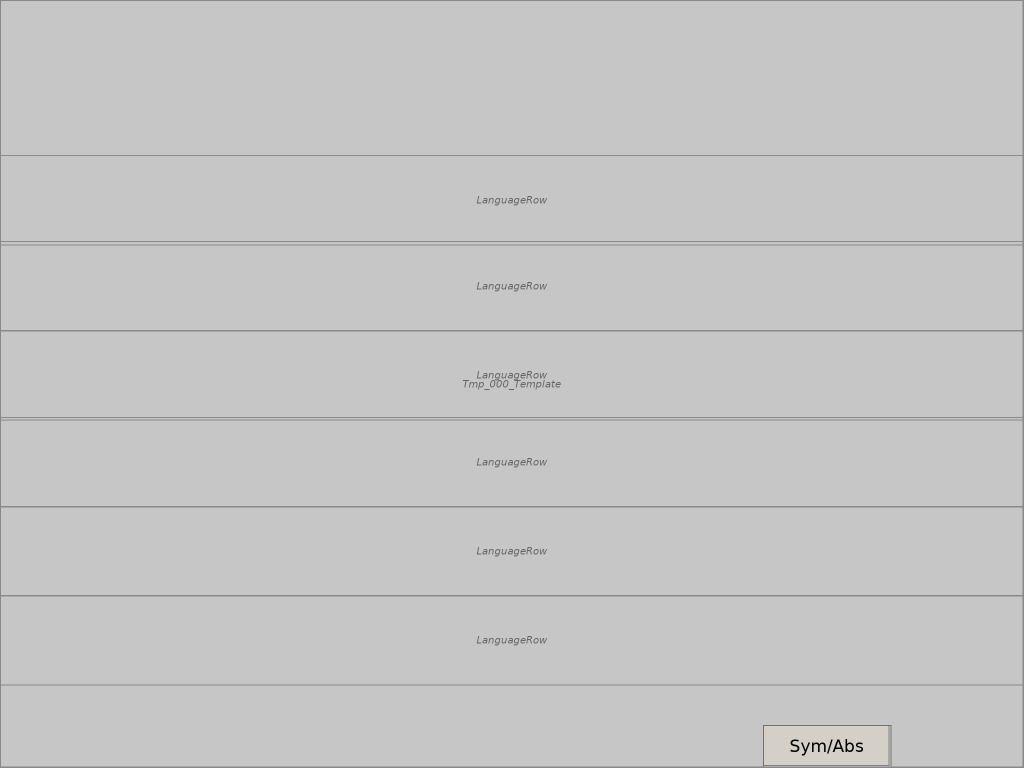
VISUALIZATION Unt_403_Language  // 1024x768
    Frame (0,0 1024x768)
        shows Tmp_000_Template(header := gHMIData.hmiHeader)
    Frame (0,155 1024x90)
        shows LanguageRow(MotionRowInstanceSingle := gHMIData.gLangRows.gMotionRow1, MotionRowButtonsSingle := gHMIData.gLangButtons.gMotionRow1btn)
    Frame (0,241 1024x90)
        shows LanguageRow(MotionRowInstanceSingle := gHMIData.gLangRows.gMotionRow2, MotionRowButtonsSingle := gHMIData.gLangButtons.gMotionRow2btn)
    Frame (0,330 1024x90)
        shows LanguageRow(MotionRowInstanceSingle := gHMIData.gLangRows.gMotionRow3, MotionRowButtonsSingle := gHMIData.gLangButtons.gMotionRow3btn)
    Frame (0,417 1024x90)
        shows LanguageRow(MotionRowInstanceSingle := gHMIData.gLangRows.gMotionRow4, MotionRowButtonsSingle := gHMIData.gLangButtons.gMotionRow4btn)
    Frame (0,506 1024x90)
        shows LanguageRow(MotionRowInstanceSingle := gHMIData.gLangRows.gMotionRow5, MotionRowButtonsSingle := gHMIData.gLangButtons.gMotionRow5btn)
    Frame (0,595 1024x90)
        shows LanguageRow(MotionRowInstanceSingle := gHMIData.gLangRows.gMotionRow6, MotionRowButtonsSingle := gHMIData.gLangButtons.gMotionRow6btn)
    Button (763,725 128x42), "Sym/Abs", colour toggle: gHMIButtons.btnAbsMode
        toggle gHMIButtons.btnAbsMode
END_VISUALIZATION

(* stored: Version 1.1.0.1, ProductVersion 3.1.4024.12
   Visu Unt_403_Language: Id {5aa6d180-b199-4212-a7f9-91e0a8fad35d} *)
